FUNCTION F_Elevationvelocity : LREAL
VAR_INPUT
	// azimuth in degrees
	azimuth:	LREAL;
	// observers latitude in degrees
	latitude:	LREAL;
END_VAR
VAR
END_VAR
VAR CONSTANT
	// Earth's angular rotation frequency in [deg/s]
	Omega: LREAL := 4.178074605556E-3;
	d2r:	LREAL := PI/180.0;
	//r2d:	LREAL := 180.0/PI;
END_VAR

//returns the rotational velocity for the azimuth in degrees per second
F_Elevationvelocity := SIN(azimuth*d2r) * COS(latitude*d2r) * Omega;

END_FUNCTION

(* stored: Version 1.1.0.1, ProductVersion 3.1.4024.9
   POU F_Elevationvelocity: Id {c42a2839-5c1e-49cc-93fc-575144a6ced3}, SpecialFunc None *)
